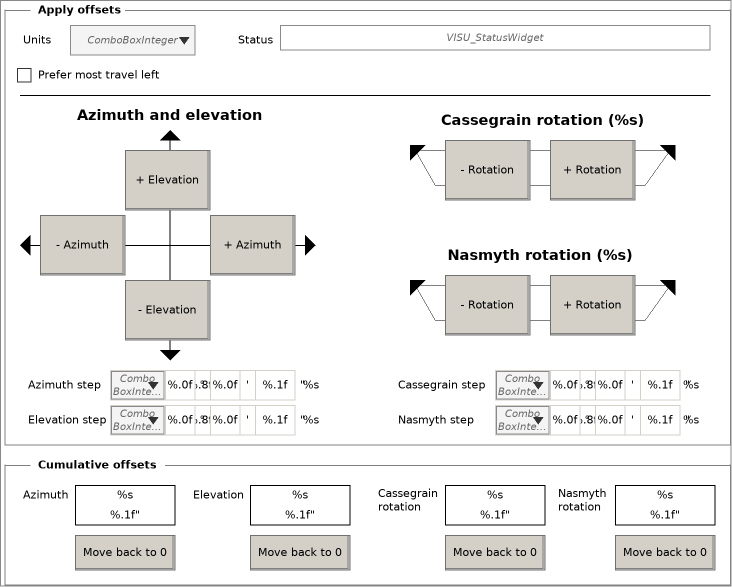
VISUALIZATION VISU_AxesManual_Offsets_AziEleRot  // 732x587
VAR_IN_OUT
	ref : Axes;
    widget : AxesManualOffsetsWidget;
END_VAR
    Polyline (125,10) (730,10) (730,445) (5,445) (5,10) (30,10)
    Polygon (670,150) (645,185) (435,185) (415,150)
    Line (170,355) (170,135)
    Line (25,245) (315,245)
    ComboBoxInteger (70,25 125x30), variable: widget.moveRelative.units, text list: 'AxesMoveProcessUnitsTextList'
    Rectangle (300,370 35x30), "%s", text variable: widget.moveRelative.unitsText, invisible if: widget.moveRelative.units = AxesMoveProcessWidgetUnits.DEGMINSEC
    Textfield (110,370 180x30), "%.8f", text variable: widget.moveRelative.field_azi_decimal, invisible if: widget.moveRelative.units = AxesMoveProcessWidgetUnits.DEGMINSEC, input disabled if: widget.moveRelative.aziDisabled
        OnMouseClick: write the text variable via VisuDialogs.Numpad
    Textfield (165,370 30x30), "%.0f", text variable: widget.moveRelative.field_azi_d, invisible if: widget.moveRelative.units <> AxesMoveProcessWidgetUnits.DEGMINSEC, input disabled if: widget.moveRelative.aziDisabled
        OnMouseClick: write the text variable via VisuDialogs.Numpad
    ComboBoxInteger (111,371 53x28), variable: widget.moveRelative.field_azi_sign, invisible if: widget.moveRelative.units <> AxesMoveProcessWidgetUnits.DEGMINSEC, input disabled if: widget.moveRelative.aziDisabled, text list: 'AxesDialogSignTextList'
    Textfield (210,370 30x30), "%.0f", text variable: widget.moveRelative.field_azi_m, invisible if: widget.moveRelative.units <> AxesMoveProcessWidgetUnits.DEGMINSEC, input disabled if: widget.moveRelative.aziDisabled
        OnMouseClick: write the text variable via VisuDialogs.Numpad
    Textfield (255,370 40x30), "%.1f", text variable: widget.moveRelative.field_azi_s, invisible if: widget.moveRelative.units <> AxesMoveProcessWidgetUnits.DEGMINSEC, input disabled if: widget.moveRelative.aziDisabled
        OnMouseClick: write the text variable via VisuDialogs.Numpad
    Label (195,370 15x30), "°", invisible if: widget.moveRelative.units <> AxesMoveProcessWidgetUnits.DEGMINSEC
    Label (240,370 15x30), "'", invisible if: widget.moveRelative.units <> AxesMoveProcessWidgetUnits.DEGMINSEC
    Label (295,370 15x30), """, invisible if: widget.moveRelative.units <> AxesMoveProcessWidgetUnits.DEGMINSEC
    Rectangle (300,405 35x30), "%s", text variable: widget.moveRelative.unitsText, invisible if: widget.moveRelative.units = AxesMoveProcessWidgetUnits.DEGMINSEC
    Textfield (110,405 180x30), "%.8f", text variable: widget.moveRelative.field_ele_decimal, invisible if: widget.moveRelative.units = AxesMoveProcessWidgetUnits.DEGMINSEC, input disabled if: widget.moveRelative.eleDisabled
        OnMouseClick: write the text variable via VisuDialogs.Numpad
    Textfield (165,405 30x30), "%.0f", text variable: widget.moveRelative.field_ele_d, invisible if: widget.moveRelative.units <> AxesMoveProcessWidgetUnits.DEGMINSEC, input disabled if: widget.moveRelative.eleDisabled
        OnMouseClick: write the text variable via VisuDialogs.Numpad
    ComboBoxInteger (111,406 53x28), variable: widget.moveRelative.field_ele_sign, invisible if: widget.moveRelative.units <> AxesMoveProcessWidgetUnits.DEGMINSEC, input disabled if: widget.moveRelative.eleDisabled, text list: 'AxesDialogSignTextList'
    Textfield (210,405 30x30), "%.0f", text variable: widget.moveRelative.field_ele_m, invisible if: widget.moveRelative.units <> AxesMoveProcessWidgetUnits.DEGMINSEC, input disabled if: widget.moveRelative.eleDisabled
        OnMouseClick: write the text variable via VisuDialogs.Numpad
    Textfield (255,405 40x30), "%.1f", text variable: widget.moveRelative.field_ele_s, invisible if: widget.moveRelative.units <> AxesMoveProcessWidgetUnits.DEGMINSEC, input disabled if: widget.moveRelative.eleDisabled
        OnMouseClick: write the text variable via VisuDialogs.Numpad
    Label (195,405 15x30), "°", invisible if: widget.moveRelative.units <> AxesMoveProcessWidgetUnits.DEGMINSEC
    Label (240,405 15x30), "'", invisible if: widget.moveRelative.units <> AxesMoveProcessWidgetUnits.DEGMINSEC
    Label (295,405 15x30), """, invisible if: widget.moveRelative.units <> AxesMoveProcessWidgetUnits.DEGMINSEC
    Rectangle (680,370 35x30), "%s", text variable: widget.moveRelative.unitsText, invisible if: widget.moveRelative.units = AxesMoveProcessWidgetUnits.DEGMINSEC
    Textfield (495,370 180x30), "%.8f", text variable: widget.moveRelative.field_roc_decimal, invisible if: widget.moveRelative.units = AxesMoveProcessWidgetUnits.DEGMINSEC, input disabled if: widget.moveRelative.rocDisabled
        OnMouseClick: write the text variable via VisuDialogs.Numpad
    Textfield (550,370 30x30), "%.0f", text variable: widget.moveRelative.field_roc_d, invisible if: widget.moveRelative.units <> AxesMoveProcessWidgetUnits.DEGMINSEC, input disabled if: widget.moveRelative.rocDisabled
        OnMouseClick: write the text variable via VisuDialogs.Numpad
    ComboBoxInteger (496,371 53x28), variable: widget.moveRelative.field_roc_sign, invisible if: widget.moveRelative.units <> AxesMoveProcessWidgetUnits.DEGMINSEC, input disabled if: widget.moveRelative.rocDisabled, text list: 'AxesDialogSignTextList'
    Textfield (595,370 30x30), "%.0f", text variable: widget.moveRelative.field_roc_m, invisible if: widget.moveRelative.units <> AxesMoveProcessWidgetUnits.DEGMINSEC, input disabled if: widget.moveRelative.rocDisabled
        OnMouseClick: write the text variable via VisuDialogs.Numpad
    Textfield (640,370 40x30), "%.1f", text variable: widget.moveRelative.field_roc_s, invisible if: widget.moveRelative.units <> AxesMoveProcessWidgetUnits.DEGMINSEC, input disabled if: widget.moveRelative.rocDisabled
        OnMouseClick: write the text variable via VisuDialogs.Numpad
    Label (580,370 15x30), "°", invisible if: widget.moveRelative.units <> AxesMoveProcessWidgetUnits.DEGMINSEC
    Label (625,370 15x30), "'", invisible if: widget.moveRelative.units <> AxesMoveProcessWidgetUnits.DEGMINSEC
    Label (680,370 15x30), """, invisible if: widget.moveRelative.units <> AxesMoveProcessWidgetUnits.DEGMINSEC
    Rectangle (680,405 35x30), "%s", text variable: widget.moveRelative.unitsText, invisible if: widget.moveRelative.units = AxesMoveProcessWidgetUnits.DEGMINSEC
    Textfield (495,405 180x30), "%.8f", text variable: widget.moveRelative.field_ron_decimal, invisible if: widget.moveRelative.units = AxesMoveProcessWidgetUnits.DEGMINSEC, input disabled if: widget.moveRelative.ronDisabled
        OnMouseClick: write the text variable via VisuDialogs.Numpad
    Textfield (550,405 30x30), "%.0f", text variable: widget.moveRelative.field_ron_d, invisible if: widget.moveRelative.units <> AxesMoveProcessWidgetUnits.DEGMINSEC, input disabled if: widget.moveRelative.ronDisabled
        OnMouseClick: write the text variable via VisuDialogs.Numpad
    ComboBoxInteger (496,406 53x28), variable: widget.moveRelative.field_ron_sign, invisible if: widget.moveRelative.units <> AxesMoveProcessWidgetUnits.DEGMINSEC, input disabled if: widget.moveRelative.ronDisabled, text list: 'AxesDialogSignTextList'
    Textfield (595,405 30x30), "%.0f", text variable: widget.moveRelative.field_ron_m, invisible if: widget.moveRelative.units <> AxesMoveProcessWidgetUnits.DEGMINSEC, input disabled if: widget.moveRelative.ronDisabled
        OnMouseClick: write the text variable via VisuDialogs.Numpad
    Textfield (640,405 40x30), "%.1f", text variable: widget.moveRelative.field_ron_s, invisible if: widget.moveRelative.units <> AxesMoveProcessWidgetUnits.DEGMINSEC, input disabled if: widget.moveRelative.ronDisabled
        OnMouseClick: write the text variable via VisuDialogs.Numpad
    Label (580,405 15x30), "°", invisible if: widget.moveRelative.units <> AxesMoveProcessWidgetUnits.DEGMINSEC
    Label (625,405 15x30), "'", invisible if: widget.moveRelative.units <> AxesMoveProcessWidgetUnits.DEGMINSEC
    Label (680,405 15x30), """, invisible if: widget.moveRelative.units <> AxesMoveProcessWidgetUnits.DEGMINSEC
    Frame (280,25 430x25)
        shows VISU_StatusWidget(widget := widget.moveRelative.actualStatus)
    Label (35,0 100x20), "Apply offsets"
    Button (125,150 85x60), "+ Elevation", input disabled if: widget.moveRelative.eleDisabled
        OnMouseClick: execute {
            ref.processes.moveRelative.request(
                units := AxesMoveUnits.DEGREES,
                azi := 0.0,
                ele := widget.moveRelative.eleDeg,
                rot := 0.0,
                roc := 0.0,
                ron := 0.0,
                doAzi := FALSE,
                doEle := TRUE,
                doRot := FALSE,
                doRoc := FALSE,
                doRon := FALSE,
                preferMostTravel := widget.preferMostTravel);
        }
    Button (125,280 85x60), "- Elevation", input disabled if: widget.moveRelative.eleDisabled
        OnMouseClick: execute {
            ref.processes.moveRelative.request(
                units := AxesMoveUnits.DEGREES,
                azi := 0.0,
                ele := -widget.moveRelative.eleDeg,
                rot := 0.0,
                roc := 0.0,
                ron := 0.0,
                doAzi := FALSE,
                doEle := TRUE,
                doRot := FALSE,
                doRoc := FALSE,
                doRon := FALSE,
                preferMostTravel := widget.preferMostTravel);
        }
    Button (210,215 85x60), "+ Azimuth", input disabled if: widget.moveRelative.aziDisabled
        OnMouseClick: execute {
            ref.processes.moveRelative.request(
                units := AxesMoveUnits.DEGREES,
                azi := widget.moveRelative.aziDeg,
                ele := 0.0,
                rot := 0.0,
                roc := 0.0,
                ron := 0.0,
                doAzi := TRUE,
                doEle := FALSE,
                doRot := FALSE,
                doRoc := FALSE,
                doRon := FALSE,
                preferMostTravel := widget.preferMostTravel);
        }
    Button (40,215 85x60), "- Azimuth", input disabled if: widget.moveRelative.aziDisabled
        OnMouseClick: execute {
            ref.processes.moveRelative.request(
                units := AxesMoveUnits.DEGREES,
                azi := -widget.moveRelative.aziDeg,
                ele := 0.0,
                rot := 0.0,
                roc := 0.0,
                ron := 0.0,
                doAzi := TRUE,
                doEle := FALSE,
                doRot := FALSE,
                doRoc := FALSE,
                doRon := FALSE,
                preferMostTravel := widget.preferMostTravel);
        }
    Label (25,370 80x30), "Azimuth step"
    Label (25,405 85x30), "Elevation step"
    Button (550,140 85x60), "+ Rotation", input disabled if: widget.moveRelative.rocDisabled
        OnMouseClick: execute {
            ref.processes.moveRelative.request(
                units := AxesMoveUnits.DEGREES,
                azi := 0.0,
                ele := 0.0,
                rot := 0.0,
                roc := widget.moveRelative.rocDeg,
                ron := 0.0,
                doAzi := FALSE,
                doEle := FALSE,
                doRot := FALSE,
                doRoc := TRUE,
                doRon := FALSE,
                preferMostTravel := widget.preferMostTravel);
        }
    Button (445,140 85x60), "- Rotation", input disabled if: widget.moveRelative.rocDisabled
        OnMouseClick: execute {
            ref.processes.moveRelative.request(
                units := AxesMoveUnits.DEGREES,
                azi := 0.0,
                ele := 0.0,
                rot := 0.0,
                roc := -widget.moveRelative.rocDeg,
                ron := 0.0,
                doAzi := FALSE,
                doEle := FALSE,
                doRot := FALSE,
                doRoc := TRUE,
                doRon := FALSE,
                preferMostTravel := widget.preferMostTravel);
        }
    Polygon (160,140) (170,130) (180,140)
    Polygon (30,255) (20,245) (30,235)
    Polygon (305,255) (315,245) (305,235)
    Polygon (160,350) (170,360) (180,350)
    Polygon (675,160) (675,145) (660,145)
    Polygon (410,160) (425,145) (410,145)
    Label (395,370 130x30), "Cassegrain step"
    Label (395,405 130x30), "Nasmyth step"
    Label (20,25 55x30), "Units"
    Label (235,25 45x30), "Status"
    Line (20,95) (710,95)
    Polygon (670,285) (645,320) (435,320) (415,285)
    Button (550,275 85x60), "+ Rotation", input disabled if: widget.moveRelative.ronDisabled
        OnMouseClick: execute {
            ref.processes.moveRelative.request(
                units := AxesMoveUnits.DEGREES,
                azi := 0.0,
                ele := 0.0,
                rot := 0.0,
                roc := 0.0,
                ron := widget.moveRelative.ronDeg,
                doAzi := FALSE,
                doEle := FALSE,
                doRot := FALSE,
                doRoc := FALSE,
                doRon := TRUE,
                preferMostTravel := widget.preferMostTravel);
        }
    Button (445,275 85x60), "- Rotation", input disabled if: widget.moveRelative.ronDisabled
        OnMouseClick: execute {
            ref.processes.moveRelative.request(
                units := AxesMoveUnits.DEGREES,
                azi := 0.0,
                ele := 0.0,
                rot := 0.0,
                roc := 0.0,
                ron := -widget.moveRelative.ronDeg,
                doAzi := FALSE,
                doEle := FALSE,
                doRot := FALSE,
                doRoc := FALSE,
                doRon := TRUE,
                preferMostTravel := widget.preferMostTravel);
        }
    Polygon (675,295) (675,280) (660,280)
    Polygon (410,295) (425,280) (410,280)
    Label (35,100 270x30), "Azimuth and elevation"
    Polyline (165,465) (730,465) (730,585) (5,585) (5,465) (30,465)
    Rectangle (75,485 100x20), "%s", text variable: widget.aziTargetOffset.dmsString
    Rectangle (75,505 100x20), "%.1f"", text variable: ref.parts.azi.targetOffset.arcseconds.value
    Button (75,535 100x35), "Move back to 0", input disabled if: widget.moveRelative.aziDisabled
        OnMouseClick: execute {
            ref.processes.moveRelative.request(
                units := AxesMoveUnits.DEGREES,
                azi := -ref.parts.azi.targetOffset.degrees.value,
                ele := 0.0,
                rot := 0.0,
                roc := 0.0,
                ron := 0.0,
                doAzi := TRUE,
                doEle := FALSE,
                doRot := FALSE,
                doRoc := FALSE,
                doRon := FALSE,
                preferMostTravel := widget.preferMostTravel);
        }
    Label (35,455 120x20), "Cumulative offsets"
    Rectangle (75,485 100x40), colour toggle: widget.moveRelative.aziDisabled
    Rectangle (250,485 100x20), "%s", text variable: widget.eleTargetOffset.dmsString
    Rectangle (250,505 100x20), "%.1f"", text variable: ref.parts.ele.targetOffset.arcseconds.value
    Button (250,535 100x35), "Move back to 0", input disabled if: widget.moveRelative.eleDisabled
        OnMouseClick: execute {
            ref.processes.moveRelative.request(
                units := AxesMoveUnits.DEGREES,
                azi := 0.0,
                ele := -ref.parts.ele.targetOffset.degrees.value,
                rot := 0.0,
                roc := 0.0,
                ron := 0.0,
                doAzi := FALSE,
                doEle := TRUE,
                doRot := FALSE,
                doRoc := FALSE,
                doRon := FALSE,
                preferMostTravel := widget.preferMostTravel);
        }
    Rectangle (250,485 100x40), colour toggle: widget.moveRelative.eleDisabled
    Rectangle (445,485 100x20), "%s", text variable: widget.rocTargetOffset.dmsString
    Rectangle (445,505 100x20), "%.1f"", text variable: ref.parts.roc.targetOffset.arcseconds.value
    Button (445,535 100x35), "Move back to 0", input disabled if: widget.moveRelative.rocDisabled
        OnMouseClick: execute {
            ref.processes.moveRelative.request(
                units := AxesMoveUnits.DEGREES,
                azi := 0.0,
                ele := 0.0,
                rot := 0.0,
                roc := -ref.parts.roc.targetOffset.degrees.value,
                ron := 0.0,
                doAzi := FALSE,
                doEle := FALSE,
                doRot := FALSE,
                doRoc := TRUE,
                doRon := FALSE,
                preferMostTravel := widget.preferMostTravel);
        }
    Rectangle (445,485 100x40), colour toggle: widget.moveRelative.rocDisabled
    Label (375,485 70x30), "Cassegrain rotation"
    Rectangle (615,485 100x20), "%s", text variable: widget.ronTargetOffset.dmsString
    Rectangle (615,505 100x20), "%.1f"", text variable: ref.parts.ron.targetOffset.arcseconds.value
    Button (615,535 100x35), "Move back to 0", input disabled if: widget.moveRelative.ronDisabled
        OnMouseClick: execute {
            ref.processes.moveRelative.request(
                units := AxesMoveUnits.DEGREES,
                azi := 0.0,
                ele := 0.0,
                rot := 0.0,
                roc := 0.0,
                ron :=  -ref.parts.ron.targetOffset.degrees.value,
                doAzi := FALSE,
                doEle := FALSE,
                doRot := FALSE,
                doRoc := FALSE,
                doRon := TRUE, preferMostTravel := widget.preferMostTravel);
        }
    Rectangle (615,485 100x40), colour toggle: widget.moveRelative.ronDisabled
    Label (555,485 60x30), "Nasmyth rotation"
    Label (20,485 55x20), "Azimuth"
    Label (190,485 55x20), "Elevation"
    Rectangle (390,240 300x30), "Nasmyth rotation (%s)", text variable: ref.config.nasmythRotatorName
    Rectangle (390,105 305x30), "Cassegrain rotation (%s)", text variable: ref.config.cassegrainRotatorName
    Checkbox (15,60 195x30), "Prefer most travel left", variable: widget.preferMostTravel
END_VISUALIZATION

(* stored: Version 1.1.0.1, ProductVersion 3.1.4019.2
   Visu VISU_AxesManual_Offsets_AziEleRot: Id {9ea7bcfc-965c-4ff7-bb70-3d95f0318305} *)
